(*	HMI variables

	This block holds all HMI variables and handles communication with the HMI
	
	2024-02 HP
		-initial
*)
{attribute 'no_explicit_call' := 'do not call this POU directly'}
FUNCTION_BLOCK HMI_TemplateMachinePart EXTENDS HMI_BaseBlock

//HMI variables that can be written to by the plc and HMI 
VAR_INPUT
	//Do not change these names, the HMI is hardcoded to use these exact names
	MAN:HMI_MAN_TemplateMachinePart;			//HMI manuals
	STS:HMI_STS_TemplateMachinePart;			//HMI statusses
	WRN:HMI_WRN_TemplateMachinePart;			//HMI warnings
	ERR:HMI_ERR_TemplateMachinePart;			//HMI errors
END_VAR

//Hmi variables that can only be written to by the HMI and read by the plc
VAR_OUTPUT PERSISTENT
	//Do not change these names, the HMI is hardcoded to use these exact names
	SP:HMI_SP_TemplateMachinePart;				//HMI setpoints
END_VAR

//this block should not be called

END_FUNCTION_BLOCK

(* stored: Version 1.1.0.1
   POU HMI_TemplateMachinePart: Id {4e896665-c713-0372-2f45-12cfc4d4d60b}, SpecialFunc None *)
